RoboDK station: LegoProject.rdk

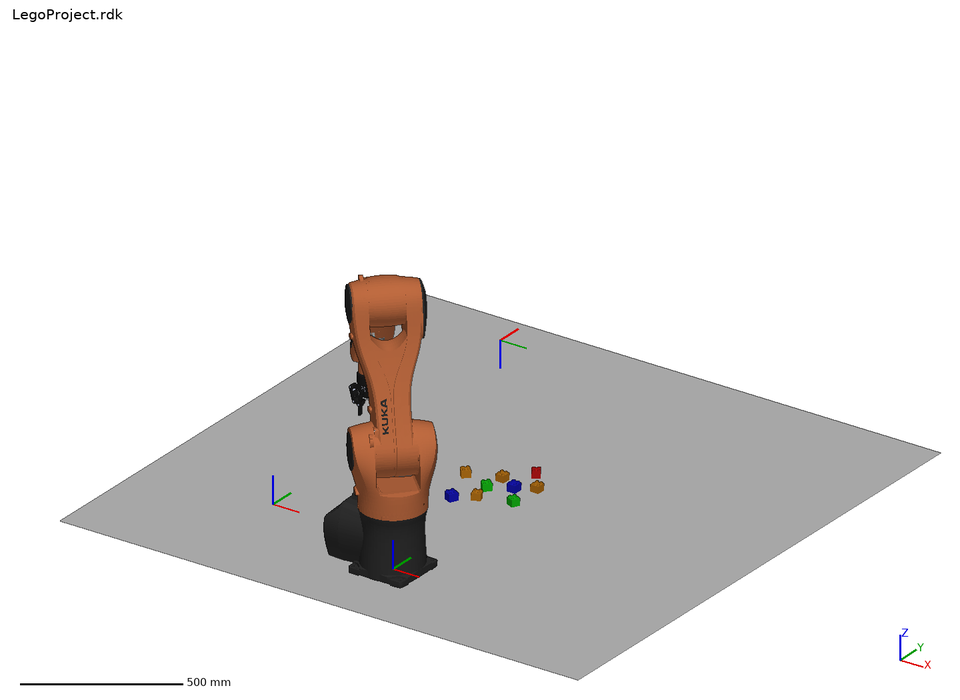
[picture v0: the station drawn from its stored meshes, robots at their saved joint values, targets as dots, program paths as lines]
Station LegoProject. Poses are relative to the parent item; angles as X-Y-Z fixed-axis rotations.
Station parameters (name, value as stored): SizeBox, 5,5,5
  - Python program StartCalib_class (listed below)
  - frame RobotBase at (-283.94, 500, 0) mm
    - object Table at (216.06, 1000, 0) mm, size 1193.8 x 965.2 x 609.6 mm, geometry from welding_table.sld
    - robot KUKA KR 6 R900 sixx: 6 axes, payload 6 kg, reach 901 mm, repeatability 0.03 mm, weight 52 kg
        modified DH rows (alpha deg, a mm, theta deg, d mm): 0, 0, 0, 400; -90, 25, 0, 0; 0, 455, -90, 0; -90, 35, 0, 420; 90, 0, 0, 0; -90, 0, 180, 80
        joint limits [-170, -190, -120, -185, -120, -350] to [170, 45, 156, 185, 120, 350]; home [0, -90, 90, 0, 0, 0]; saved at [-134.119, -71.916, 122.553, 180, -39.363, -134.119]
      - tool Gripper, TCP at (0, 0, 150) mm, size 134.4 x 157.6 x 75 mm
    - frame WorkSpace at (-560, 160, 0) mm
      - frame CameraRef at (500, 500, 500) mm, rotated rx 180 ry 0 rz 90 deg
      - object Green 1 at (606.06, 420, 0) mm, rotated rx 0 ry 0 rz -115 deg, size 30 x 30 x 30 mm, geometry from Green.sld
      - object Green 2 at (476.06, 460, 0) mm, rotated rx 0 ry 0 rz -40 deg, size 30 x 30 x 30 mm, geometry from Green.sld
      - object grayPlane at (500, 500, 0) mm, size 1940.1 x 1940.1 x 0 mm, geometry from grayPlane.stl
      - object RedCalib at (546.06, 490, 0) mm, size 30 x 30 x 30 mm, geometry from Red.sld
      - object YellowCalib at (646.06, 530, 0) mm, size 30 x 30 x 30 mm, geometry from Yellow.sld
      - object BlueCalib at (460, 480, 0) mm, size 32 x 32 x 32 mm, geometry from Blue.fbx
      - object GreenCalib at (606.06, 420, 0) mm, rotated rx 0 ry 0 rz -115 deg, size 30 x 30 x 30 mm, geometry from Green.sld
      - object Yellow 3 at (490.14, 389.86, 0) mm, rotated rx 0 ry 0 rz 20 deg, size 30 x 30 x 30 mm, geometry from Yellow.sld
      - object Blue 1 at (429.32, 340.48, 0) mm, rotated rx 0 ry 0 rz -25 deg, size 32 x 32 x 32 mm, geometry from Blue.fbx
      - object Yellow 1 at (369.72, 500.19, 0) mm, rotated rx 0 ry 0 rz 45.61 deg, size 30 x 30 x 30 mm, geometry from Yellow.sld
      - object Blue 2 at (550.1, 500.61, 0) mm, rotated rx 0 ry 0 rz 89.46 deg, size 32 x 32 x 32 mm, geometry from Blue.fbx
      - object Yellow 4 at (480.21, 539.97, 0) mm, rotated rx 0 ry 0 rz -0.34 deg, size 30 x 30 x 30 mm, geometry from Yellow.sld
      - object Red 1 at (550.18, 619.7, 0) mm, rotated rx 0 ry 0 rz 34.55 deg, size 30 x 30 x 30 mm, geometry from Red.sld
      - object Yellow 2 at (610, 540, 0) mm, rotated rx 0 ry 0 rz 89.46 deg, size 30 x 30 x 30 mm, geometry from Yellow.sld

--- Python program StartCalib_class ---
from robolink import *    # API to communicate with RoboDK
from robodk import *      # robodk robotics toolbox
import cv2 as cv
import numpy as np
from matplotlib import pyplot as plt
import argparse
from numpy import loadtxt
from numpy import genfromtxt
from numpy import savetxt

# Any interaction with RoboDK must be done through RDK: So those have to be written in order to communicate with RoboDk
RDK = Robolink()
RDK.Cam2D_Close() #Closes any preopened camera view

# get the robot by name:
robot = RDK.Item('KUKA KR 6 R900 sixx', ITEM_TYPE_ROBOT)

# get the targets references by name:
home = RDK.Item('Home')
target = RDK.Item('Plane')

# get the pose of the target (4x4 matrix representing position and orientation):
poseref = target.Pose() # This gives the position of the target reference but as a mat type, but it's currently not used anywhere

# move the robot to home, then to the the : Uncheck to try
#robot.MoveJ(home)
#robot.MoveJ(poseref)
#print(robot.ConnectedState())
#"{} and {}".format("Robot connection:", robot.ConnectedState())


#get the size of the lego bricks from the user
PARAM_SIZE_BOX = 'SizeBox'
SIZE_BOX = RDK.getParam('SizeBox')
size_box = RDK.getParam(PARAM_SIZE_BOX)

size_box_input = mbox('Enter the size of the box in mm [L,W,H]', entry=size_box)
if size_box_input:
    RDK.setParam(PARAM_SIZE_BOX, size_box_input)
else:
    raise Exception('Operation cancelled by user')

#print(size_box_input)
robot.setJoints([90,-90,90,0,0,0])
#------------------------------------------------------------
#Select the camera and settings
cameraf=RDK.ItemUserPick('Select the Camera location (reference, tool or object)')
cam_id = RDK.Cam2D_Add(cameraf, 'FOCAL_LENGHT=6 FOV=38 FAR_LENGHT=2100 SIZE=640x480 BG_COLOR=black LIGHT_SPECULAR=white')

#-----------------------------------------------------------------------------------
#Get the height or whatever of the brick
SIZE_BOX_XYZ = [float(x.replace(' ','')) for x in SIZE_BOX.split(',')]
SIZE_BOX_Z=SIZE_BOX_XYZ[2]
#--------------------------------------------------------------------------
#Take a snapshot of the cameraRef view then save it
path= RDK.getParam('PATH_OPENSTATION')
RDK.Cam2D_Snapshot(path + "/image.png", cam_id)
#----------------------------------------------------------------------
#This is to locate the brick in the image, so change the location
#       to where you save your image in the previous step
imagepath=r'E:\OneDrive\OneDrive - Aalborg Universitet\AAU\8th semester\P8\DGCNN\SemesterProject_843\Lego\image.png'
image1=cv.imread(imagepath)
lower_color_bounds = np.array([0,250,0])
upper_color_bounds = np.array([0,255,80])


#cv.imshow('original_img',image1)
cv.imwrite(path+"/originalimage.jpg",image1)

#COLOR DETECTION --> Thresholds: HSV
def DetectColor(image,lower_boundary,upper_boundary):
    mask = cv.inRange(image, lower_boundary, upper_boundary)
    color_image = cv.bitwise_and(image,image, mask= mask)
    return color_image

def ComputeSlope(image,image2):
    #h,s,v = cv.split(image)
    closing = cv.morphologyEx(image, cv.MORPH_CLOSE, np.ones((5,5)))
    closing = cv.Canny(closing, 50, 200, None, 3)
    closing = cv.dilate(closing,(3,3),iterations = 1)
    cv.imshow("canny",closing)
    lines = cv.HoughLinesP(closing,1,np.pi/180,10,10,10)
    #print("Found lines:",len(lines))
    if lines is not None:
        for line in lines:
            for x1,y1,x2,y2 in line:
                cv.line(image2,(x1,y1),(x2,y2),(0,0,0),2)
                slope = (y2-y1)/(x2-x1)
                slope = math.atan(slope)
                slope = math.degrees(slope)
                return slope
                #print("Slope is:",slope)

hsv_img = cv.cvtColor(image1, cv.COLOR_BGR2HSV)
red_color = DetectColor(hsv_img,lower_boundary = np.array([-15,90,220]), upper_boundary = np.array([15,255,255]))
green_color = DetectColor(hsv_img,lower_boundary = np.array([138/2-15,90,220]), upper_boundary = np.array([138/2+15,255,255]))
yellow_color = DetectColor(hsv_img,lower_boundary = np.array([57/2-15,90,220]), upper_boundary = np.array([59/2+15,255,255]))
#-------------------------------------------------------
#Find the location for each point
h,s,v= cv.split(red_color)
firstGray=cv.cvtColor(red_color,cv.COLOR_HSV2BGR)
firstGray=cv.cvtColor(red_color,cv.COLOR_BGR2GRAY)
firstGray = cv.bitwise_not(firstGray)
detector=cv.SimpleBlobDetector_create()
cv.imshow("firstgray",firstGray)
keypoints = detector.detect(firstGray)
firstGray = cv.bitwise_not(firstGray)
#im_with_keypoints=cv.drawKeypoints(firstGray,keypoints,np.array([]),(255,255,255),cv.DRAW_MATCHES_FLAGS_DRAW_RICH_KEYPOINTS)
im_with_keypoints=firstGray
cv.imshow("imwithkeypoints",im_with_keypoints)
red_brick_loc=[]
for i in keypoints:
    x = i.pt[0] #i is the index of the blob you want to get the position
    y = i.pt[1]
    red_brick_loc.append([[y],[x],[1]])
print(red_brick_loc)
cv.imshow("ima",im_with_keypoints)
#-------------------------------------------------------
#Extract the patches
patch_center = np.array([red_brick_loc[1][0], red_brick_loc[1][1]])# the location of the patch
print (patch_center)
patch_scale = 0.18# the area to be patched

smaller_dim = np.min(im_with_keypoints.shape[0:2])
patch_size = int(patch_scale * smaller_dim)
patch_x = int(patch_center[0] - patch_size / 2.)
patch_y = int(patch_center[1] - patch_size / 2.)
patch_image = im_with_keypoints[patch_x:patch_x+patch_size, patch_y:patch_y+patch_size]
cv.imshow('patch_image', patch_image)
patch_image = cv.morphologyEx(patch_image, cv.MORPH_CLOSE, np.ones((5,5)))
# show image and patch
cv.imshow('image', im_with_keypoints)
#cv.imshow('patch_image', patch_image)
#-------------------------------------------------------
#Resize the image
scale_percent = 220 # percent of original size
width = int(patch_image.shape[1] * scale_percent / 100)
height = int(patch_image.shape[0] * scale_percent / 100)
dim = (width, height)
# resize image
patch_image = cv.resize(patch_image, dim, interpolation = cv.INTER_AREA)
cv.imshow("Resized image", patch_image)
#-------------------------------------------------------

slope = ComputeSlope(patch_image,image1)
print(slope)
cv.imshow("OriginalImage",image1)
target= patch_center
robot.setJoints([0,0,0,0,90,slope])
approach = target.Pose()*transl(0,0,-100)


#mtx is the cameras intrinsic and extrinsic parameters
#mtx = genfromtxt('E:\OneDrive\OneDrive - Aalborg Universitet\AAU\8th semester\RobotVision\Miniproject\Lego\mtx.csv', delimiter=',')
#rvecs = genfromtxt('E:\OneDrive\OneDrive - Aalborg Universitet\AAU\8th semester\RobotVision\Miniproject\Lego\ecs.csv', delimiter=',')
#print(brick_loc)
"""
x1 = brick_loc[3][0][0]
y1 = brick_loc[3][1][0]
x1c = 0.0
y1c = 0.0

x2 = brick_loc[2][0][0]
y2 = brick_loc[2][1][0]
x2c = 1000.0
y2c = 0.0

x3 = brick_loc[1][0][0]
y3 = brick_loc[1][1][0]
x3c = 0.0
y3c = 1000.0

x4 = brick_loc[0][0][0]
y4 = brick_loc[0][1][0]
x4c = 1000
y4c = 1000

a = np.array(
    [[x1,0,x2,0,x3,0,x4,0],
    [y1,0,y2,0,y3,0,y4,0],
    [1,0,1,0,1,0,1,0],
    [0,x1,0,x2,0,x3,0,x4],
    [0,y1,0,y2,0,y3,0,y4],
    [0,1,0,1,0,1,0,1],
    [-x1*x1c,-x1*y1c,-x2*x2c,-x2*y2c,-x3*x3c,-x3*y3c,-x4*x4c,-x4*y4c],
    [-y1*x1c,-y1*y1c,-y2*x2c,-y2*y2c,-y3*x3c,-y3*y3c,-y4*x4c,-y4*x4c]])

a = np.transpose(a)

b = [x1c,y1c,x2c,y2c,x3c,y3c,x4c,y4c]
 """
def mapping(x,y,d):
    xC = ((d[0]*x)+(d[1]*y)+d[2])/((d[6]*x)+(d[7]*y)+1)
    yC = ((d[3]*x)+(d[4]*y)+d[5])/((d[6]*x)+(d[7]*y)+1)
    return xC,yC

#d=np.linalg.solve(a,b)
#savetxt(r'E:\OneDrive\OneDrive - Aalborg Universitet\AAU\8th semester\P8\DGCNN\SemesterProject_843\Lego\d.csv',d, delimiter='')

""" testX,testY= mapping(x4,y4,d)

print(testX,testY) """

#print(np.allclose(np.dot(a, x), b))



if cv.waitKey():
    RDK.Cam2D_Close() #Closes any preopened camera view
